RoboDK station: maros_v0.1.rdk

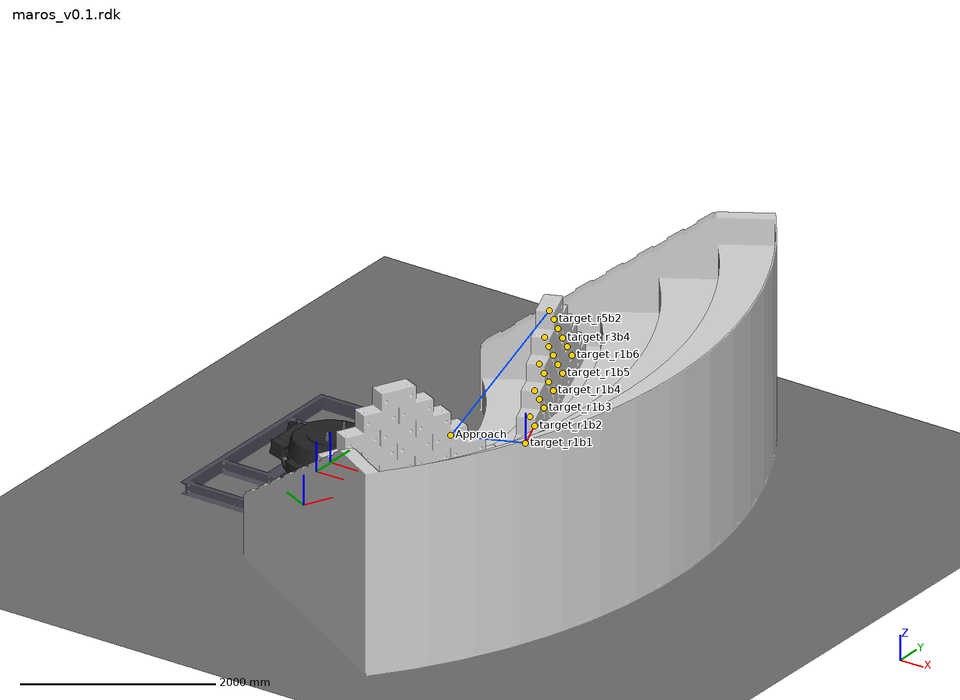
[picture v0: the station drawn from its stored meshes, robots at their saved joint values, targets as dots, program paths as lines]
Station maros_v0.1 (saved by RoboDK 5.4.1). Poses are relative to the parent item; angles as X-Y-Z fixed-axis rotations.
  - folder assets
    - object Floor at (0, 0, 0) mm, size 9000 x 9000 x 0 mm, geometry from Floor.sld
    - object Stairs_v1 at (-2520, 0, 0) mm, size 3922.2 x 7408.9 x 2302 mm, geometry from Stairs_v1.3ds
    - object Frame at (0, 0, 0) mm, size 2000 x 2500 x 199.8 mm, geometry from Frame.stp
  - frame KUKA KR 210-2 Base at (0, 0, 140) mm
    - robot KUKA KR 210-2: 6 axes, payload 210 kg, reach 2700 mm, repeatability 0.06 mm, weight 1267 kg
        joint limits [-185, -146, -119, -350, -125, -350] to [185, 0, 155, 350, 125, 350]; home [0, -90, 90, 0, 0, 0]; saved at [57.559, -53.201, 78.303, -123.6, 40.25, 131.04]
      - tool NEMO_ASM-v2, TCP at (50, 0, 430) mm, size 350 x 350 x 427.5 mm, geometry from NEMO_ASM-v2.stp
    - frame Table 1 at (2270, 238.94, 760) mm, rotated rx 0 ry 0 rz 112 deg
      - target target_r1b1 (Cartesian target) at (0, 0, 0) mm, rotated rx 0 ry 90 rz -90 deg; joints [2.067, -52.896, 108.321, -145.978, 60.263, 161.487] of KUKA KR 210-2
      - target target_r1b2 (Cartesian target) at (420, 0, 0) mm, rotated rx 0 ry 90 rz -90 deg; joints [-11.873, -56.834, 117.553, -162.781, 61.827, 171.675] of KUKA KR 210-2
      - target target_r1b3 (Cartesian target) at (840, 0, 0) mm, rotated rx 0 ry 90 rz -90 deg; joints [-27.87, -58.059, 120.514, -180.981, 62.458, 180.454] of KUKA KR 210-2
      - target target_r1b4 (Cartesian target) at (1260, 0, 0) mm, rotated rx 0 ry 90 rz -90 deg; joints [-43.736, -56.543, 116.857, -199.092, 61.689, 189.322] of KUKA KR 210-2
      - target target_r1b5 (Cartesian target) at (1680, 0, 0) mm, rotated rx 0 ry 90 rz -90 deg; joints [-57.379, -52.32, 106.997, -215.696, 60.08, 199.716] of KUKA KR 210-2
      - target target_r1b6 (Cartesian target) at (2100, 0, 0) mm, rotated rx 0 ry 90 rz -90 deg; joints [-68.079, -45.403, 91.45, -230.448, 58.454, 212.354] of KUKA KR 210-2
      - target target_r2b1 (Cartesian target) at (210, 0, 200) mm, rotated rx 0 ry 90 rz -90 deg; joints [-4.556, -63.685, 112.198, -151.127, 52.247, 161.345] of KUKA KR 210-2
      - target target_r2b2 (Cartesian target) at (630, 0, 200) mm, rotated rx 0 ry 90 rz -90 deg; joints [-19.73, -67.105, 118.287, -170.702, 51.551, 174.187] of KUKA KR 210-2
      - target target_r2b3 (Cartesian target) at (1050, 0, 200) mm, rotated rx 0 ry 90 rz -90 deg; joints [-35.975, -66.907, 117.939, -191.483, 51.597, 187.192] of KUKA KR 210-2
      - target target_r2b4 (Cartesian target) at (1470, 0, 200) mm, rotated rx 0 ry 90 rz -90 deg; joints [-50.915, -63.129, 111.192, -210.8, 52.343, 200.011] of KUKA KR 210-2
      - target target_r2b5 (Cartesian target) at (1890, 0, 200) mm, rotated rx 0 ry 90 rz -90 deg; joints [-63.09, -56.325, 98.57, -227.315, 53.258, 212.968] of KUKA KR 210-2
      - target target_r3b1 (Cartesian target) at (420, 0, 400) mm, rotated rx 0 ry 90 rz -90 deg; joints [-11.873, -73.433, 112.651, -156.851, 41.591, 162.268] of KUKA KR 210-2
      - target target_r3b2 (Cartesian target) at (840, 0, 400) mm, rotated rx 0 ry 90 rz -90 deg; joints [-27.87, -75.428, 115.47, -181.352, 40.05, 181.035] of KUKA KR 210-2
      - target target_r3b3 (Cartesian target) at (1260, 0, 400) mm, rotated rx 0 ry 90 rz -90 deg; joints [-43.736, -72.971, 111.985, -205.532, 41.92, 199.566] of KUKA KR 210-2
      - target target_r3b4 (Cartesian target) at (1680, 0, 400) mm, rotated rx 0 ry 90 rz -90 deg; joints [-57.379, -66.672, 102.456, -225.072, 45.585, 215.054] of KUKA KR 210-2
      - target target_r4b1 (Cartesian target) at (640, 0, 600) mm, rotated rx 0 ry 90 rz -90 deg; joints [-20.114, -81.144, 109.759, -165.847, 29.364, 167.605] of KUKA KR 210-2
      - target target_r4b2 (Cartesian target) at (1060, 0, 600) mm, rotated rx 0 ry 90 rz -90 deg; joints [-36.355, -80.757, 109.291, -199.028, 29.906, 196.644] of KUKA KR 210-2
      - target target_r4b3 (Cartesian target) at (1480, 0, 600) mm, rotated rx 0 ry 90 rz -90 deg; joints [-51.24, -75.656, 102.814, -224.608, 35.776, 218.67] of KUKA KR 210-2
      - target target_r5b1 (Cartesian target) at (860, 0, 800) mm, rotated rx 0 ry 90 rz -90 deg; joints [-28.649, -85.852, 103.546, -185.41, 17.768, 185.153] of KUKA KR 210-2
      - target target_r5b2 (Cartesian target) at (1280, 0, 800) mm, rotated rx 0 ry 90 rz -90 deg; joints [-44.447, -82.727, 100.045, -226.556, 24.391, 223.879] of KUKA KR 210-2
      - target target_r6 (Cartesian target) at (1070, 0, 1000) mm, rotated rx 0 ry 90 rz -90 deg; joints [-36.734, -87.365, 94.367, -234.601, 11.971, 234.004] of KUKA KR 210-2
      - object r6 at (1070, 0, 1000) mm, size 400 x 200 x 210 mm, geometry from brick_Origin.sld
      - object r1b1 at (0, 0, 0) mm, size 400 x 200 x 210 mm, geometry from brick_Origin.sld
        - object r1b2 at (420, 0, 0) mm, size 400 x 200 x 210 mm, geometry from brick_Origin.sld
          - object r1b3 at (420, 0, 0) mm, size 400 x 200 x 210 mm, geometry from brick_Origin.sld
            - object r1b4 at (420, 0, 0) mm, size 400 x 200 x 210 mm, geometry from brick_Origin.sld
              - object r1b5 at (420, 0, 0) mm, size 400 x 200 x 210 mm, geometry from brick_Origin.sld
                - object r1b6 at (420, 0, 0) mm, size 400 x 200 x 210 mm, geometry from brick_Origin.sld
      - object r2b1 at (210, 0, 200) mm, size 400 x 200 x 210 mm, geometry from brick_Origin.sld
        - object r2b2 at (420, 0, 0) mm, size 400 x 200 x 210 mm, geometry from brick_Origin.sld
          - object r2b3 at (420, 0, 0) mm, size 400 x 200 x 210 mm, geometry from brick_Origin.sld
            - object r2b4 at (420, 0, 0) mm, size 400 x 200 x 210 mm, geometry from brick_Origin.sld
              - object r2b5 at (420, 0, 0) mm, size 400 x 200 x 210 mm, geometry from brick_Origin.sld
      - object r3b1 at (420, 0, 400) mm, size 400 x 200 x 210 mm, geometry from brick_Origin.sld
        - object r3b2 at (420, 0, 0) mm, size 400 x 200 x 210 mm, geometry from brick_Origin.sld
          - object r3b3 at (420, 0, 0) mm, size 400 x 200 x 210 mm, geometry from brick_Origin.sld
            - object r3b4 at (420, 0, 0) mm, size 400 x 200 x 210 mm, geometry from brick_Origin.sld
      - object r4b1 at (640, 0, 600) mm, size 400 x 200 x 210 mm, geometry from brick_Origin.sld
        - object r4b2 at (420, 0, 0) mm, size 400 x 200 x 210 mm, geometry from brick_Origin.sld
          - object r4b3 at (420, 0, 0) mm, size 400 x 200 x 210 mm, geometry from brick_Origin.sld
      - object r5b1 at (860, 0, 800) mm, size 400 x 200 x 210 mm, geometry from brick_Origin.sld
        - object r5b2 at (420, 0, 0) mm, size 400 x 200 x 210 mm, geometry from brick_Origin.sld
    - frame Table 2 at (1260, -2281.06, 784.46) mm, rotated rx 0 ry 0 rz 65 deg
      - object r6 at (1070, 0, 1000) mm, size 400 x 200 x 210 mm, geometry from brick_Origin.sld
      - object r1b1 at (0, 0, 0) mm, size 400 x 200 x 210 mm, geometry from brick_Origin.sld
        - object r1b2 at (420, 0, 0) mm, size 400 x 200 x 210 mm, geometry from brick_Origin.sld
          - object r1b3 at (420, 0, 0) mm, size 400 x 200 x 210 mm, geometry from brick_Origin.sld
            - object r1b4 at (420, 0, 0) mm, size 400 x 200 x 210 mm, geometry from brick_Origin.sld
              - object r1b5 at (420, 0, 0) mm, size 400 x 200 x 210 mm, geometry from brick_Origin.sld
                - object r1b6 at (420, 0, 0) mm, size 400 x 200 x 210 mm, geometry from brick_Origin.sld
      - object r2b1 at (210, 0, 200) mm, size 400 x 200 x 210 mm, geometry from brick_Origin.sld
        - object r2b2 at (420, 0, 0) mm, size 400 x 200 x 210 mm, geometry from brick_Origin.sld
          - object r2b3 at (420, 0, 0) mm, size 400 x 200 x 210 mm, geometry from brick_Origin.sld
            - object r2b4 at (420, 0, 0) mm, size 400 x 200 x 210 mm, geometry from brick_Origin.sld
              - object r2b5 at (420, 0, 0) mm, size 400 x 200 x 210 mm, geometry from brick_Origin.sld
      - object r3b1 at (420, 0, 400) mm, size 400 x 200 x 210 mm, geometry from brick_Origin.sld
        - object r3b2 at (420, 0, 0) mm, size 400 x 200 x 210 mm, geometry from brick_Origin.sld
          - object r3b3 at (420, 0, 0) mm, size 400 x 200 x 210 mm, geometry from brick_Origin.sld
            - object r3b4 at (420, 0, 0) mm, size 400 x 200 x 210 mm, geometry from brick_Origin.sld
      - object r4b1 at (640, 0, 600) mm, size 400 x 200 x 210 mm, geometry from brick_Origin.sld
        - object r4b2 at (420, 0, 0) mm, size 400 x 200 x 210 mm, geometry from brick_Origin.sld
          - object r4b3 at (420, 0, 0) mm, size 400 x 200 x 210 mm, geometry from brick_Origin.sld
      - object r5b1 at (860, 0, 800) mm, size 400 x 200 x 210 mm, geometry from brick_Origin.sld
        - object r5b2 at (420, 0, 0) mm, size 400 x 200 x 210 mm, geometry from brick_Origin.sld
    - frame Base at (0, -250.97, 0) mm
      - target Approach (Cartesian target) at (1566.96, 158.82, 784.46) mm, rotated rx 0 ry 90 rz 0 deg; joints [5.802, -70.303, 150.121, 185.894, 79.87, -181.04] of KUKA KR 210-2
  - program Pick and place (10 instructions, listed below)
  - Python program Main (listed below)
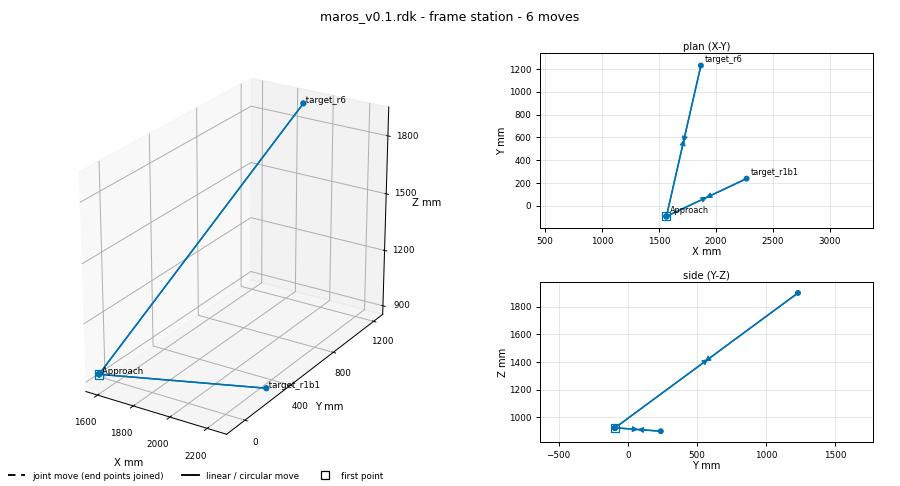
[picture p0: tool path of maros_v0.1.rdk in frame station, 6 of 6 moves have a stored position in this frame; points joined in program order, loops and branches not executed]

--- program Pick and place (robot KUKA KR 210-2) ---
  Set Frame: Table 1
  Set Tool: NEMO_ASM-v2
  Set speed (200.0 mm/s)
  MoveJ (Approach)
  MoveL (target_top) -> target target_r6
  MoveL (Approach)
  Set Ref.: Table 2
  MoveJ (Approach)
  MoveL (target_r1b1)
  MoveL (Approach)

--- Python program Main ---
# Type help("robodk.robolink") or help("robodk.robomath") for more information
# Press F5 to run the script
# Documentation: https://robodk.com/doc/en/RoboDK-API.html
# Reference:     https://robodk.com/doc/en/PythonAPI/robodk.html
# Note: It is not required to keep a copy of this file, your Python script is saved with your RDK project
from robodk import robolink    # RoboDK API
from robodk import robomath    # Robot toolbox

# The following 2 lines keep your code compatible with older versions or RoboDK:
from robodk import *      # RoboDK API
from robolink import *    # Robot toolbox

# Link to RoboDK
RDK = robolink.Robolink()
robot = RDK.Item('KUKA KR 210-2')

frame1 = RDK.Item('Table 1')
frame2 = RDK.Item('Table 2')
base = RDK.Item('Base')

pairList = [
    ['r6','r1b1'],
    ['r5b2','r1b2'],
    ['r5b1','r1b3'],
    ['r4b3','r1b4'],
    ['r4b2','r1b5'],
    ['r4b1','r1b6'],
    ['r3b4','r2b1'],
    ['r3b3','r2b2'],
    ['r3b2','r2b3'],
    ['r3b1','r2b4'],
    ['r2b5','r2b5'],
    ['r2b4','r3b1'],
    ['r2b3','r3b2'],
    ['r2b2','r3b3'],
    ['r2b1','r3b4'],
    ['r1b6','r4b1'],
    ['r1b5','r4b2'],
    ['r1b4','r4b3'],
    ['r1b3','r5b1'],
    ['r1b2','r5b2'],
    ['r1b1','r6'],
]

def moveWithOffset(target_pose, offset):
    xyz_ref = target_pose.Pos()

    x = xyz_ref[0] + offset[0]
    y = xyz_ref[1] + offset[1]
    z = xyz_ref[2] + offset[2]

    target_pose.setPos([x,y,z])
    robot.MoveL(target_pose)
    return target_pose

def moveToBase():
    robot.setPoseFrame(base)

    target = RDK.Item('Approach')
    target_pose = target.Pose()
    robot.MoveL(target_pose)

def placeBrick(target_name):
    robot.setSpeed(200)

    target = RDK.Item(f'target_{target_name}')
    target_pose = target.Pose()

    hovered_pos = moveWithOffset(target_pose, [0,0,400])
    robot.setSpeed(50)
    placed_pos = moveWithOffset(hovered_pos, [0,0,-400])
    robot.setSpeed(25)
    release_pos = moveWithOffset(placed_pos, [0,0,-10])
    robot.setSpeed(200)
    safe_pos = moveWithOffset(release_pos, [0,600,0])


def pickBrick(target_name):
    robot.setSpeed(200)

    target = RDK.Item(f'target_{target_name}')
    target_pose = target.Pose()

    approach_pose = moveWithOffset(target_pose, [0,200,0])
    robot.setSpeed(50)
    insert_pose = moveWithOffset(approach_pose, [0,-500,0])
    robot.setSpeed(100)
    lift_pose = moveWithOffset(insert_pose, [0,0,300])
    robot.setSpeed(200)
    safe_pose = moveWithOffset(lift_pose, [0,600,0])

def runMain(frame):
    frameMain = frame1 if frame else frame2
    frameAlter = frame2 if frame else frame1

    for i in pairList:
        robot.setPoseFrame(frameMain)
        pickBrick(i[0])
        moveToBase()
        robot.setPoseFrame(frameAlter)
        placeBrick(i[1])
        moveToBase()

    robot.RunInstruction('Program_Done')
    runMain(not frame)

runMain(True)
